(* PLC project LED-Identifikation.project, CODESYS CODESYS V3.5 SP21 Patch 1 *)
(* stored: creationDateTime 2026-09-30T16:31:38.7257111, modificationDateTime 2026-09-30T14:39:44.6045366 *)

PROGRAM PLC_PRG
  VAR
    fbUserLED : WagoAppAppLED.FbAppLED_SetStatic;
    stStatus : WagoAppAppLED.FbResult;
    tonBlink : TON;
    xLED : BOOL := FALSE;
  END_VAR

            fbUserLED(
    xEnable := TRUE,
    eLedID := WagoAppAppLED.eLedID.AppLED_5,
    eLedColor := WagoAppAppLED.eLedColor.Green,
    oStatus => stStatus
);
          
END_PROGRAM
